FUNCTION_BLOCK InductionMotor IMPLEMENTS I_Motor
VAR_INPUT
END_VAR
VAR_OUTPUT
END_VAR
VAR
	fRunning : BOOL;
END_VAR

{warning 'add method implementation '}
METHOD Start : BOOL
fRunning := TRUE;
Start := fRunning;
END_METHOD

{warning 'add method implementation '}
METHOD Stop : BOOL
fRunning := FALSE;
Stop := fRunning;
END_METHOD

END_FUNCTION_BLOCK

(* stored: Version 1.1.0.1, ProductVersion 3.1.4024.16
   POU InductionMotor: Id {5fdebe78-7443-4306-9eb8-872870658c14}, SpecialFunc None
   Method Start: Id {f4a3ebe4-7b7c-44ea-9055-2c88dc1b1d9e}
   Method Stop: Id {b4a101f8-95f3-4e2f-a624-61d7c9362075} *)
